Staubli VAL3: PriseEnMain.dtx

mdesc mNomSpeed
jointRx jInit
jointRx jDest
pointRx pCarre1 = {fatherId=world[0]}
pointRx pCarre2 = {fatherId=world[0]}
pointRx pCarre4 = {fatherId=world[0]}
pointRx pCarre3 = {fatherId=world[0]}
